(* IEC 61131-3 sources: plc_generation_empirical_study/datasets/_archive/native_profile_v4_20260810/tasks/C01_H01_four_level_priority, 2 files *)

(* ---- interface.st ---- *)
FUNCTION_BLOCK C01_H01_four_level_priority
VAR_INPUT
    Info : BOOL;
    Warning : BOOL;
    Trip : BOOL;
    Emergency : BOOL;
    Suppress : BOOL;
END_VAR
VAR_OUTPUT
    Active : BOOL;
    Level : INT;
END_VAR
END_FUNCTION_BLOCK

(* ---- reference.st ---- *)
FUNCTION_BLOCK C01_H01_four_level_priority
VAR_INPUT
    Info : BOOL;
    Warning : BOOL;
    Trip : BOOL;
    Emergency : BOOL;
    Suppress : BOOL;
END_VAR
VAR_OUTPUT
    Active : BOOL;
    Level : INT;
END_VAR

IF Emergency THEN
    Level := 4;
    Active := TRUE;
ELSIF Suppress THEN
    Level := 0;
    Active := FALSE;
ELSIF Trip THEN
    Level := 3;
    Active := TRUE;
ELSIF Warning THEN
    Level := 2;
    Active := TRUE;
ELSIF Info THEN
    Level := 1;
    Active := TRUE;
ELSE
    Level := 0;
    Active := FALSE;
END_IF;

END_FUNCTION_BLOCK
